// TIA Portal V15.1 export
// export: Created 2024-05-17T05:38:53.9168564Z, ExportSetting WithDefaults, DisplayName Totally Integrated Automation Portal, DisplayVersion V15.1 Update 5, DisplayName TIA Portal Openness, DisplayVersion V15.1 Update 5, DisplayName SINAMICS Startdrive Advanced, DisplayVersion V15.1, DisplayName G130, G150, S120, S150, SINAMICS MV, S210, DisplayVersion V15.1, DisplayName G110M, G120, G120C, G120D, G120P, DisplayVersion V15.1, DisplayName STEP 7 Professional, DisplayVersion V15.1 Update 5, DisplayName STEP 7 Safety, DisplayVersion V15.1, DisplayName WinCC Professional, DisplayVersion V15.1 Update 5, DisplayName SIMATIC Visualization Architect, DisplayVersion V15.1
FUNCTION_BLOCK "LVIDSRFID"   // FB1203, SCL
{ S7_Optimized_Access := 'TRUE' }
VERSION : 0.1
// stored: AutoNumber false, IsIECCheckEnabled false, IsRetainMemResEnabled false, MemoryReserve 100, SetENOAutomatically False, UDAEnableTagReadback false
   VAR_INPUT
      I_OutOfUse { ExternalAccessible := 'False'; ExternalVisible := 'False'; ExternalWritable := 'False'} : Bool;   // Module out of use
      C_AntennaTriggOnTime { ExternalAccessible := 'False'; ExternalVisible := 'False'; ExternalWritable := 'False'} : DInt := 3000;   // Default 3s
      C_AntennaTriggOffTime { ExternalAccessible := 'False'; ExternalVisible := 'False'; ExternalWritable := 'False'} : DInt := 500;   // Default 500ms
      I_AntennaStatus { ExternalAccessible := 'False'; ExternalVisible := 'False'; ExternalWritable := 'False'} : Bool;   // Antenna status
      I_StartRead { ExternalAccessible := 'False'; ExternalVisible := 'False'; ExternalWritable := 'False'} : Bool;   // On edge, start tag read
      I_InitTagEn { ExternalAccessible := 'False'; ExternalVisible := 'False'; ExternalWritable := 'False'} : Bool := FALSE;   // Init tag enabled
      I_StartInitTag { ExternalAccessible := 'False'; ExternalVisible := 'False'; ExternalWritable := 'False'} : Bool;   // On edge, start initialisation
      I_BodyIDInitTag { ExternalAccessible := 'False'; ExternalVisible := 'False'; ExternalWritable := 'False'} : DWord;   // Body identifier for init function
      I_BodyType1InitTag { ExternalAccessible := 'False'; ExternalVisible := 'False'; ExternalWritable := 'False'} : DWord;   // BodyType1
      I_PopIDInitTag { ExternalAccessible := 'False'; ExternalVisible := 'False'; ExternalWritable := 'False'} : UDInt;   // Spare Data / PopID
      I_PopIDSuffixInitTag { ExternalAccessible := 'False'; ExternalVisible := 'False'; ExternalWritable := 'False'} : Char;   // PopID suffix
      I_PopTypeInitTag { ExternalAccessible := 'False'; ExternalVisible := 'False'; ExternalWritable := 'False'} : UDInt;   // Pop identifier
      I_ResetAlarm { ExternalAccessible := 'False'; ExternalVisible := 'False'; ExternalWritable := 'False'} : Bool;   // Reset alarm
   END_VAR
   VAR_OUTPUT
      O_AntennaTrigg { ExternalAccessible := 'False'; ExternalVisible := 'False'; ExternalWritable := 'False'} : Bool;   // to antenna - start read
      O_Busy { ExternalAccessible := 'False'; ExternalVisible := 'False'; ExternalWritable := 'False'} : Bool;   // Busy
      O_ReadOK { ExternalAccessible := 'False'; ExternalVisible := 'False'; ExternalWritable := 'False'} : Bool;   // RFID read OK
      O_ReadNOK { ExternalAccessible := 'False'; ExternalVisible := 'False'; ExternalWritable := 'False'} : Bool;   // RFID read NOK
      O_InitTagBusy { ExternalAccessible := 'False'; ExternalVisible := 'False'; ExternalWritable := 'False'} : Bool;   // Tag init busy
      O_InitTagOK { ExternalAccessible := 'False'; ExternalVisible := 'False'; ExternalWritable := 'False'} : Bool;   // Tag init OK
      O_InitTagNOK { ExternalAccessible := 'False'; ExternalVisible := 'False'; ExternalWritable := 'False'} : Bool;   // Tag init NOK
      O_ReplaceTagBusy { ExternalAccessible := 'False'; ExternalVisible := 'False'; ExternalWritable := 'False'} : Bool;
      O_ReplaceTagOK { ExternalAccessible := 'False'; ExternalVisible := 'False'; ExternalWritable := 'False'} : Bool;   // Replace tag - OK
      O_ReplaceTagNOK { ExternalAccessible := 'False'; ExternalVisible := 'False'; ExternalWritable := 'False'} : Bool;   // Replace tag - NOK
      O_Status { ExternalAccessible := 'False'; ExternalVisible := 'False'; ExternalWritable := 'False'} : Int;   // Status code
      O_Alarm { ExternalAccessible := 'False'; ExternalVisible := 'False'; ExternalWritable := 'False'} : Bool;   // Alarm C / Alarm
   END_VAR
   VAR_IN_OUT
      IO_VIDS : "VIDS";   // For internal use only
      IO_VEMData : "VEMData";   // From master module
      IO_Alarm : "Alarm";   // Alarm
      H_RFID : "H_LVIDSRFID";
      H_HMI : "H_HMI";
   END_VAR
   VAR
      i { ExternalAccessible := 'False'; ExternalVisible := 'False'; ExternalWritable := 'False'} : Int;   // Index
      Reset { ExternalAccessible := 'False'; ExternalVisible := 'False'; ExternalWritable := 'False'} : Bool;
      ReadOK { ExternalAccessible := 'False'; ExternalVisible := 'False'; ExternalWritable := 'False'} : Bool;
      ReadNOK { ExternalAccessible := 'False'; ExternalVisible := 'False'; ExternalWritable := 'False'} : Bool;
      InitTagOK { ExternalAccessible := 'False'; ExternalVisible := 'False'; ExternalWritable := 'False'} : Bool;
      InitTagNOK { ExternalAccessible := 'False'; ExternalVisible := 'False'; ExternalWritable := 'False'} : Bool;
      ReplaceTagOK { ExternalAccessible := 'False'; ExternalVisible := 'False'; ExternalWritable := 'False'} : Bool;
      ReplaceTagNOK { ExternalAccessible := 'False'; ExternalVisible := 'False'; ExternalWritable := 'False'} : Bool;
      StartReplaceTagMem { ExternalAccessible := 'False'; ExternalVisible := 'False'; ExternalWritable := 'False'} : Bool;
      StartInitMem { ExternalAccessible := 'False'; ExternalVisible := 'False'; ExternalWritable := 'False'} : Bool;
      btnForceReadEdg { ExternalAccessible := 'False'; ExternalVisible := 'False'; ExternalWritable := 'False'} : Bool;
      btnForceReadPls { ExternalAccessible := 'False'; ExternalVisible := 'False'; ExternalWritable := 'False'} : Bool;
      btnInitTagByBodyIdEdg { ExternalAccessible := 'False'; ExternalVisible := 'False'; ExternalWritable := 'False'} : Bool;
      btnInitTagByBodyIdPls { ExternalAccessible := 'False'; ExternalVisible := 'False'; ExternalWritable := 'False'} : Bool;
      btnInitTagByBodyType1Edg { ExternalAccessible := 'False'; ExternalVisible := 'False'; ExternalWritable := 'False'} : Bool;
      btnInitTagByBodyType1Pls { ExternalAccessible := 'False'; ExternalVisible := 'False'; ExternalWritable := 'False'} : Bool;
      btnInitTagByPopIdEdg { ExternalAccessible := 'False'; ExternalVisible := 'False'; ExternalWritable := 'False'} : Bool;
      btnInitTagByPopIdPls { ExternalAccessible := 'False'; ExternalVisible := 'False'; ExternalWritable := 'False'} : Bool;
      btnRplcTagByMixNbrEdg { ExternalAccessible := 'False'; ExternalVisible := 'False'; ExternalWritable := 'False'} : Bool;
      btnRplcTagByMixNbrPls { ExternalAccessible := 'False'; ExternalVisible := 'False'; ExternalWritable := 'False'} : Bool;
      btnRplcTagByMixNbrEnable { ExternalAccessible := 'False'; ExternalVisible := 'False'; ExternalWritable := 'False'} : Word;
      btnRplcTagByTagIDEdg { ExternalAccessible := 'False'; ExternalVisible := 'False'; ExternalWritable := 'False'} : Bool;
      btnRplcTagByTagIDPls { ExternalAccessible := 'False'; ExternalVisible := 'False'; ExternalWritable := 'False'} : Bool;
      btnRplcTagByTagIDEnable { ExternalAccessible := 'False'; ExternalVisible := 'False'; ExternalWritable := 'False'} : Word;
      btnRplcTagByBodyIdEdg { ExternalAccessible := 'False'; ExternalVisible := 'False'; ExternalWritable := 'False'} : Bool;
      btnRplcTagByBodyIdPls { ExternalAccessible := 'False'; ExternalVisible := 'False'; ExternalWritable := 'False'} : Bool;
      btnRplcTagByBodyIdEnable { ExternalAccessible := 'False'; ExternalVisible := 'False'; ExternalWritable := 'False'} : Word;
      btnRplcTagByPopIDEdg { ExternalAccessible := 'False'; ExternalVisible := 'False'; ExternalWritable := 'False'} : Bool;
      btnRplcTagByPopIDPls { ExternalAccessible := 'False'; ExternalVisible := 'False'; ExternalWritable := 'False'} : Bool;
      btnRplcTagByPopIDEnable { ExternalAccessible := 'False'; ExternalVisible := 'False'; ExternalWritable := 'False'} : Word;
      GetVEMDataByRFIDBeginReq1 { ExternalAccessible := 'False'; ExternalVisible := 'False'; ExternalWritable := 'False'} : Bool;
      GetVEMDataByRFIDBeginReq2 { ExternalAccessible := 'False'; ExternalVisible := 'False'; ExternalWritable := 'False'} : Bool;
      GetVEMDataByRFIDBeginReq3 { ExternalAccessible := 'False'; ExternalVisible := 'False'; ExternalWritable := 'False'} : Bool;
      InteractEnable { ExternalAccessible := 'False'; ExternalVisible := 'False'; ExternalWritable := 'False'} : Bool;   // Interactions enabled
      Status { ExternalAccessible := 'False'; ExternalVisible := 'False'; ExternalWritable := 'False'} : Int;
      TriggOnTimerElapsed { ExternalAccessible := 'False'; ExternalVisible := 'False'; ExternalWritable := 'False'} : Bool;   // Antenna trigger - On
      AntennaTriggOnTimeAct { ExternalAccessible := 'False'; ExternalVisible := 'False'; ExternalWritable := 'False'} : DInt;
      TriggerOffTimerElapsed { ExternalAccessible := 'False'; ExternalVisible := 'False'; ExternalWritable := 'False'} : Bool;   // Antenna trigger - Off
      AntennaTriggOffTimeAct { ExternalAccessible := 'False'; ExternalVisible := 'False'; ExternalWritable := 'False'} : DInt;
      AntennaTrigg { ExternalAccessible := 'False'; ExternalVisible := 'False'; ExternalWritable := 'False'} : Bool;
      AntennaTriggCntr { ExternalAccessible := 'False'; ExternalVisible := 'False'; ExternalWritable := 'False'} : Int;   // Antenna trigger - Counter
      AntennaStatus { ExternalAccessible := 'False'; ExternalVisible := 'False'; ExternalWritable := 'False'} : Int;
      StartReadEdg { ExternalAccessible := 'False'; ExternalVisible := 'False'; ExternalWritable := 'False'} : Bool;
      StartReadPls { ExternalAccessible := 'False'; ExternalVisible := 'False'; ExternalWritable := 'False'} : Bool;
      StartInitTagEdg { ExternalAccessible := 'False'; ExternalVisible := 'False'; ExternalWritable := 'False'} : Bool;
      StartInitTagPls { ExternalAccessible := 'False'; ExternalVisible := 'False'; ExternalWritable := 'False'} : Bool;
      Alarm { ExternalAccessible := 'False'; ExternalVisible := 'False'; ExternalWritable := 'False'} : Bool;
      BodyIdMemReplaceTag { ExternalAccessible := 'False'; ExternalVisible := 'False'; ExternalWritable := 'False'} : DWord;
      MixNbrMemReplaceTag { ExternalAccessible := 'False'; ExternalVisible := 'False'; ExternalWritable := 'False'} : DWord;
      PopIdMemReplaceTag { ExternalAccessible := 'False'; ExternalVisible := 'False'; ExternalWritable := 'False'} : DWord;
      PopIdSuffixMemReplaceTag { ExternalAccessible := 'False'; ExternalVisible := 'False'; ExternalWritable := 'False'} : Char;
      PopTypeMemReplaceTag { ExternalAccessible := 'False'; ExternalVisible := 'False'; ExternalWritable := 'False'} : DWord;
      TagIdMem { ExternalAccessible := 'False'; ExternalVisible := 'False'; ExternalWritable := 'False'} : DWord;
      TagIdMemReplaceTag { ExternalAccessible := 'False'; ExternalVisible := 'False'; ExternalWritable := 'False'} : DWord;
      TagIdMemReplaceTagStr { ExternalAccessible := 'False'; ExternalVisible := 'False'; ExternalWritable := 'False'} : String[7];
      BodyIDMemInit { ExternalAccessible := 'False'; ExternalVisible := 'False'; ExternalWritable := 'False'} : DWord;
      BodyType1MemInit { ExternalAccessible := 'False'; ExternalVisible := 'False'; ExternalWritable := 'False'} : DWord;
      PopIDMemInit { ExternalAccessible := 'False'; ExternalVisible := 'False'; ExternalWritable := 'False'} : DWord;
      PopIDSuffixMemInit { ExternalAccessible := 'False'; ExternalVisible := 'False'; ExternalWritable := 'False'} : Char;
      PopTypeMemInit { ExternalAccessible := 'False'; ExternalVisible := 'False'; ExternalWritable := 'False'} : DWord;
      StartTriggOnTimer { ExternalAccessible := 'False'; ExternalVisible := 'False'; ExternalWritable := 'False'} : Bool;   // Trigger on timer - Start
      StartTriggOffTimer { ExternalAccessible := 'False'; ExternalVisible := 'False'; ExternalWritable := 'False'} : Bool;   // Trigger off timer - Start
      TempDiv { ExternalAccessible := 'False'; ExternalVisible := 'False'; ExternalWritable := 'False'} : DInt;   // Temporary divider
      TempDInt { ExternalAccessible := 'False'; ExternalVisible := 'False'; ExternalWritable := 'False'} : DInt;
      TempReal { ExternalAccessible := 'False'; ExternalVisible := 'False'; ExternalWritable := 'False'} : Real;
      _TriggOnTmr { ExternalAccessible := 'False'; ExternalVisible := 'False'; ExternalWritable := 'False'; S7_SetPoint := 'True'} : "LTimer";   // FB / Trigger on timer
      _TriggOffTmr { ExternalAccessible := 'False'; ExternalVisible := 'False'; ExternalWritable := 'False'; S7_SetPoint := 'True'} : "LTimer";   // FB / Trigger off timer
   END_VAR
   VAR CONSTANT
      TAG_ID_LENGTH_MAX : Int := 7;
      CMD_INIT_TAG : DWord := 2003;   // Command code - Init tag
      CMD_REPLACE_TAG : DWord := 2002;   // Command code - Replace tag
      ANTENNA_TRIGG_CNTR_MAX : Int := 3;   // Maximum amount of triggers
      STATUS_000 : Int;   // Status 000 : No action
      STATUS_001 : Int := 1;   // Status 001 : Success
      STATUS_002 : Int := 2;   // Status 002 : Busy
      STATUS_MINUS_001 : Int := -1;   // Status - 001 : No signal from RFID antenna
      STATUS_MINUS_002 : Int := -2;   // Status - 002 : Tag read error
      STATUS_MINUS_008 : Int := -12;   // Status - 008 : Sequence overtime
      STATUS_MINUS_100 : Int := -100;   // Status - 100 : TagId does not exist
      OFF : Word := 16#0000;   // HMI animation - No animation
      VISIBLE : Word := 16#0001;   // HMI animation - Visible
      ENABLE : Word := 16#0002;   // HMI animation - Enable
      COLOUR_DEFAULT : Word := 16#0000;   // HMI animation - Default colour
      COLOUR_RED : Word := 16#0010;   // HMI animation - Colour red
      COLOUR_GREEN : Word := 16#0020;   // HMI animation - Colour green
      COLOUR_BLUE : Word := 16#0040;   // HMI animation - Colour blue
      COLOUR_WHITE : Word := 16#0080;   // HMI animation - Colour white
      SECTION_HMI : Bool := TRUE;
      SECTION_OUTPUTS : Bool := TRUE;
   END_VAR
BEGIN
   (******************************************************************************
    Changelog

       17W23D1 18:00H PMo
       - Conversion from FBD TO SCL

    List OF authors

       Company : Volvo Cars Gent
       Name    : Patrick Moreau (PMo)
       E-mail  : patrick.moreau@volvocars.com
       Tel.    : +32 9 2503165

    Description

       This module is part OF the VIDS suite and is used to read, initialize and 
       replace the RFID.
       To use this module, VIDSMaster is required

    ******************************************************************************)

   (******************************************************************************)
   (* Alarm                                                                      *)
   (******************************************************************************)
   IF NOT #I_AntennaStatus AND NOT #IO_VIDS.GetVEMDataByRFID.Running AND FALSE THEN        //Check antenna
       #Status := #STATUS_MINUS_001;   //No signal from RFID antenna
   END_IF;
   IF #I_AntennaStatus AND #Status = #STATUS_MINUS_001 AND FALSE THEN
       #Status := #STATUS_000;
   END_IF;

   (******************************************************************************)
   (* Create pulses                                                              *)
   (******************************************************************************)

   //Start read - Create pulse
   #StartReadPls := #I_StartRead AND NOT #StartReadEdg;
   #StartReadEdg := #I_StartRead;

   //< Force read > button - Create pulse
   #btnForceReadPls := #H_RFID.H_btnForceRead <> 0 AND NOT #btnForceReadEdg;
   #btnForceReadEdg := #H_RFID.H_btnForceRead <> 0;

   //Start init - Create pulse
   #StartInitTagPls := #I_StartInitTag AND NOT #StartInitTagEdg;
   #StartInitTagEdg := #I_StartInitTag;

   // < Start Init tag BY BodyID > button - Create pulse
   #btnInitTagByBodyIdPls := (#H_RFID.H_btnInitTagByBodyId <> 0) AND NOT #btnInitTagByBodyIdEdg;
   #btnInitTagByBodyIdEdg := (#H_RFID.H_btnInitTagByBodyId <> 0);

   // < Start Init tag BY BodyType1 > button - Create pulse
   #btnInitTagByBodyType1Pls := (#H_RFID.H_btnInitTagByBodyType1 <> 0) AND NOT #btnInitTagByBodyType1Edg;
   #btnInitTagByBodyType1Edg := (#H_RFID.H_btnInitTagByBodyType1 <> 0);

   // < Start Init tag BY PopID > button - Create pulse
   #btnInitTagByPopIdPls := (#H_RFID.H_btnInitTagByPopId <> 0) AND NOT #btnInitTagByPopIdEdg;
   #btnInitTagByPopIdEdg := (#H_RFID.H_btnInitTagByPopId <> 0);

   //< Replace Tag BY TagID > button - Create pulse
   #btnRplcTagByTagIDPls := #H_RFID.H_btnRplcTagByTagID <> 0 AND NOT #btnRplcTagByTagIDEdg;
   #btnRplcTagByTagIDEdg := #H_RFID.H_btnRplcTagByTagID <> 0;

   //< Replace Tag BY BodyID > button - Create pulse
   #btnRplcTagByBodyIdPls := #H_RFID.H_btnRplcTagByBodyId <> 0 AND NOT #btnRplcTagByBodyIdEdg;
   #btnRplcTagByBodyIdEdg := #H_RFID.H_btnRplcTagByBodyId <> 0;

   //< Replace Tag BY Mixnumber > button - Create pulse
   #btnRplcTagByMixNbrPls := #H_RFID.H_btnRplcTagByMIxNbr <> 0 AND NOT #btnRplcTagByMixNbrEdg;
   #btnRplcTagByMixNbrEdg := #H_RFID.H_btnRplcTagByMIxNbr <> 0;

   //< Replace Tag BY PopId > button - Create pulse
   #btnRplcTagByPopIDPls := #H_RFID.H_btnRplcTagByPopId <> 0 AND NOT #btnRplcTagByPopIDEdg;
   #btnRplcTagByPopIDEdg := #H_RFID.H_btnRplcTagByPopId <> 0;

   (******************************************************************************)
   (* Get VEM data by RFID - Begin request                                       *)
   (******************************************************************************)

   //By Read
   #GetVEMDataByRFIDBeginReq1 := #I_AntennaStatus AND (#StartReadPls OR #btnForceReadPls);

   //By Replace tag
   IF  #btnRplcTagByTagIDPls THEN
       #TagIdMemReplaceTag := #H_RFID.H_txtTagIDRplcTag;
       #BodyIdMemReplaceTag := 0;
       #MixNbrMemReplaceTag := 0;
       #PopIdMemReplaceTag := 0;
       #PopIdSuffixMemReplaceTag := ' ';
       #PopTypeMemReplaceTag := 0;
       #StartReplaceTagMem := TRUE;
   ELSIF  #btnRplcTagByBodyIdPls THEN
       #TagIdMemReplaceTag := 0;
       #BodyIdMemReplaceTag := #H_RFID.H_txtBodyIDRplcTag;
       #MixNbrMemReplaceTag := 0;
       #PopIdMemReplaceTag := 0;
       #PopIdSuffixMemReplaceTag := ' ';
       #PopTypeMemReplaceTag := 0;
       #StartReplaceTagMem := TRUE;
   ELSIF  #btnRplcTagByMixNbrPls THEN
       #TagIdMemReplaceTag :=0;
       #BodyIdMemReplaceTag := 0;
       #MixNbrMemReplaceTag := #H_RFID.H_txtMixNbrRplcTag;
       #PopIdMemReplaceTag := 0;
       #PopIdSuffixMemReplaceTag := ' ';
       #PopTypeMemReplaceTag := 0;
       #StartReplaceTagMem := TRUE;
   ELSIF  #btnRplcTagByPopIDPls THEN
       #TagIdMemReplaceTag := 0;
       #BodyIdMemReplaceTag := 0;
       #MixNbrMemReplaceTag := 0;
       #PopIdMemReplaceTag := #H_RFID.H_txtPopIDRplcTag;
       #PopIdSuffixMemReplaceTag := #H_RFID.H_txtPopIDSuffixRplcTag;
       #PopTypeMemReplaceTag := #H_RFID.H_txtPopTypeRplcTag;
       #StartReplaceTagMem := TRUE;
   END_IF;
   #GetVEMDataByRFIDBeginReq2 := #btnRplcTagByTagIDPls OR #btnRplcTagByBodyIdPls OR #btnRplcTagByMixNbrPls OR #btnRplcTagByPopIDPls;

   //By Init tag
   IF  #StartInitTagPls THEN
       IF #I_BodyIDInitTag <> 0 THEN
           #BodyIDMemInit := #I_BodyIDInitTag;
           #BodyType1MemInit := 0;
           #PopIDMemInit := 0;
           #PopIDSuffixMemInit := ' ';
           #PopTypeMemInit := 0;
       ELSIF #I_BodyType1InitTag <> 0 THEN
           #BodyIDMemInit := 0;
           #PopIDMemInit := 0;
           #PopIDSuffixMemInit := ' ';
           #PopTypeMemInit := 0;
           #BodyType1MemInit := #I_BodyType1InitTag;
       ELSIF #I_PopIDInitTag <> 0 THEN
           #BodyIDMemInit := 0;
           #BodyType1MemInit := 0;
           #PopIDMemInit := #I_PopIDInitTag;
           #PopIDSuffixMemInit := #I_PopIDSuffixInitTag;
           #PopTypeMemInit := #I_PopTypeInitTag;
       END_IF;
       #StartInitMem := TRUE;
   ELSIF  #btnInitTagByBodyIdPls THEN
       #BodyIDMemInit := #H_RFID.H_txtBodyIDInitTag;
       #BodyType1MemInit := 0;
       #PopIDMemInit := 0;
       #PopIDSuffixMemInit := ' ';
       #PopTypeMemInit := 0;
       #StartInitMem := TRUE;
   ELSIF #I_AntennaStatus AND #btnInitTagByBodyType1Pls THEN
       #BodyIDMemInit := 0;
       #PopIDMemInit := 0;
       #PopIDSuffixMemInit := ' ';
       #PopTypeMemInit := 0;
       #BodyType1MemInit := #H_RFID.H_txtBodyType1InitTag;
       #StartInitMem := TRUE;
   ELSIF #I_AntennaStatus AND #btnInitTagByPopIdPls THEN
       #BodyIDMemInit := 0;
       #BodyType1MemInit := 0;
       #PopIDMemInit := #H_RFID.H_txtPopIdInitTag;
       #PopIDSuffixMemInit := #H_RFID.H_txtPopIdSuffixInitTag;
       #PopTypeMemInit := #H_RFID.H_txtPopTypeInitTag;
       #StartInitMem := TRUE;
   END_IF;

   #GetVEMDataByRFIDBeginReq3 := #StartInitTagPls OR #btnInitTagByBodyIdPls OR #btnInitTagByBodyType1Pls OR #btnInitTagByPopIdPls;

   //Begin request - Summary
   #IO_VIDS.GetVEMDataByRFID.BeginReq := #IO_VIDS.PartPres  AND
   (#GetVEMDataByRFIDBeginReq1 OR #GetVEMDataByRFIDBeginReq2 OR #GetVEMDataByRFIDBeginReq3) AND NOT 
   #IO_VIDS.GetVEMDataByRFID.Running;

   //Reset when not part present
   IF NOT #IO_VIDS.PartPres THEN

       #StartReplaceTagMem := FALSE;
       #StartInitMem := FALSE;

   END_IF;

   #Reset := NOT #IO_VIDS.PartPres OR #IO_VIDS.GetVEMDataByRFID.BeginReq OR #IO_VIDS.InitTag.BeginReq OR #IO_VIDS.ReplaceTag.BeginReq;

   IF  #Reset THEN



       #ReadOK := FALSE;
       #ReadNOK := FALSE;
       #InitTagOK := FALSE;
       #InitTagNOK := FALSE;
       #ReplaceTagOK := FALSE;
       #ReplaceTagNOK := FALSE;
       #AntennaStatus := 0;
       #Status := 0;

   END_IF;

   (******************************************************************************)
   (* Get VEM data by RFID - Begin                                               *)
   (******************************************************************************)

   //Activate antenna
   IF #IO_VIDS.GetVEMDataByRFID.OkBegin THEN
       #Status := #STATUS_002;             //Set Status busy

       #AntennaTriggCntr := 0;             //Reset antenna trigger Counter
       #StartTriggOnTimer := TRUE;         //Start trigger
   END_IF;

   //Step 0 On Active - Get VEM Data - Begin
   #IO_VIDS.GetVEMDataByRFID.Begin := #IO_VIDS.GetVEMDataByRFID.OkBegin;

   (******************************************************************************)
   (* Get VEM data by RFID - Antenna triggering                                  *)
   (******************************************************************************)

   IF NOT #I_AntennaStatus THEN
       #StartTriggOnTimer := FALSE;
       #StartTriggOffTimer := FALSE;
   END_IF;

   //Antenna Trigger on timer
   #_TriggOnTmr(I_StartTimer := #StartTriggOnTimer,
                I_HoldTimer := FALSE,
                I_MaxTimerValue := #C_AntennaTriggOnTime,
                O_TimerResult => #TriggOnTimerElapsed,
                O_TimerValue => #AntennaTriggOnTimeAct);

   //Start off timer
   IF #TriggOnTimerElapsed THEN
       #StartTriggOnTimer := FALSE;
       #StartTriggOffTimer := TRUE;
   END_IF;

   //Antenna Trigger off timer
   #_TriggOffTmr(I_StartTimer := #StartTriggOffTimer,
                 I_HoldTimer := FALSE,
                 I_MaxTimerValue := #C_AntennaTriggOffTime,
                 O_TimerResult => #TriggerOffTimerElapsed,
                 O_TimerValue => #AntennaTriggOffTimeAct);

   //Restart trigger timer
   IF #TriggerOffTimerElapsed THEN
       #AntennaTriggCntr := #AntennaTriggCntr + 1;
       IF #AntennaTriggCntr < #ANTENNA_TRIGG_CNTR_MAX THEN
           #StartTriggOffTimer := FALSE;
           #StartTriggOnTimer := TRUE;
       ELSE
           #StartTriggOnTimer := FALSE;
           #StartTriggOffTimer := FALSE;
           #AntennaStatus := #STATUS_MINUS_002;
       END_IF;
   END_IF;

   //Antenna Trigger
   #AntennaTrigg := #StartTriggOnTimer AND NOT #TriggOnTimerElapsed AND #I_AntennaStatus;

   (******************************************************************************)
   (* Get VEM data by RFID - Finish                                              *)
   (******************************************************************************)

   //Make sure we create a pulse
   #IO_VIDS.ReplaceTag.BeginReq := FALSE;
   #IO_VIDS.InitTag.BeginReq := FALSE;

   //Get VEMData by RFID - Finished
   IF #IO_VIDS.GetVEMDataByRFID.Finished THEN

       //Antenna status has priority
       IF #AntennaStatus < 0 THEN
           #Status := #AntennaStatus;
       ELSE
           #Status := #IO_VIDS.GetVEMDataByRFID.Status;
       END_IF;

       //Read OK or NOK
       IF #Status = 1 THEN
           #ReadOK := True;
       ELSE
           #ReadNOK := True;
       END_IF;

       //Replace tag
       IF #StartReplaceTagMem THEN
           #StartReplaceTagMem := FALSE;
           IF #Status <> #STATUS_MINUS_002 THEN
               #TagIdMem := #IO_VIDS.VEMData.Identification;
               #IO_VIDS.ReplaceTag.BeginReq := TRUE;       //Replace tag - Begin request
           END_IF;

       //Init tag
       ELSIF #StartInitMem THEN
           #StartInitMem := FALSE;
           IF #Status <> #STATUS_MINUS_002 THEN
               #TagIdMem := #IO_VIDS.VEMData.Identification;
               #IO_VIDS.InitTag.BeginReq := TRUE;
           END_IF;
       END_IF;

   END_IF;

   (******************************************************************************)
   (* Replace tag - Begin & Finished                                             *)
   (******************************************************************************)

   IF #IO_VIDS.ReplaceTag.OkBegin THEN

       #Status := #STATUS_002;             //Set Status busy
       #IO_VIDS.VEMData.CommandCode := #CMD_REPLACE_TAG;
       #IO_VIDS.VEMData.Identification := #TagIdMem;

       IF #TagIdMemReplaceTag <> 0 THEN
           //TagId in specificdata
           #TempDInt := DWORD_TO_DINT(#TagIdMemReplaceTag);
           #TempReal := DINT_TO_REAL(#TAG_ID_LENGTH_MAX-1);
           #TempDiv := REAL_TO_DINT(10 ** #TempReal);
           FOR #i := 0 TO (#TAG_ID_LENGTH_MAX-1) DO
               #IO_VIDS.SpecificDataInit[#i] := DINT_TO_CHAR(#TempDInt / #TempDiv + 48);
               #TempDInt := #TempDInt MOD #TempDiv;
               #TempDiv := #TempDiv / 10;
           END_FOR;
           #IO_VIDS.VEMData.SpecificDataLength := DINT_TO_DWORD(#TAG_ID_LENGTH_MAX);
       ELSE
           #IO_VIDS.VEMData.BodyID := #BodyIdMemReplaceTag;
           #IO_VIDS.VEMData.MixNumber := #MixNbrMemReplaceTag;
           #IO_VIDS.VEMData.PopID := #PopIdMemReplaceTag;
           #IO_VIDS.VEMData.PopIDSuffix := #PopIdSuffixMemReplaceTag;
           #IO_VIDS.VEMData.PopType := #PopTypeMemReplaceTag;
           #IO_VIDS.VEMData.SpecificDataLength := 0;
       END_IF;

   ELSIF #IO_VIDS.ReplaceTag.Finished THEN
       #Status := #IO_VIDS.ReplaceTag.Status;
       IF #Status = 1 THEN
           #ReplaceTagOK := True;
       ELSE
           #ReplaceTagNOK := True;
       END_IF;
   END_IF;

   #IO_VIDS.ReplaceTag.Begin := #IO_VIDS.ReplaceTag.OkBegin;

   (******************************************************************************)
   (* Init tag - Begin & Finished                                                *)
   (******************************************************************************)

   IF #IO_VIDS.InitTag.OkBegin THEN

       #Status := #STATUS_002;             //Set Status busy
       #IO_VIDS.VEMData.Identification := #TagIdMem;
       #IO_VIDS.VEMData.BodyID := #BodyIDMemInit;
       #IO_VIDS.VEMData.BodyType1 := #BodyType1MemInit;
       #IO_VIDS.VEMData.PopID := #PopIDMemInit;
       #IO_VIDS.VEMData.PopIDSuffix := #PopIDSuffixMemInit;
       #IO_VIDS.VEMData.PopType := #PopTypeMemInit;

       #IO_VIDS.VEMData.CommandCode := #CMD_INIT_TAG;

   ELSIF #IO_VIDS.InitTag.Finished THEN
       #Status := #IO_VIDS.InitTag.Status;
       IF #Status = 1 THEN
           #InitTagOK := True;
       ELSE
           #InitTagNOK := True;
       END_IF;
   END_IF;

   #IO_VIDS.InitTag.Begin := #IO_VIDS.InitTag.OkBegin;

   (******************************************************************************)
   (* Alarm = status <0                                                          *)
   (******************************************************************************)
   IF #Status < 0 THEN
       #Alarm := TRUE;
   ELSE
       #Alarm := false;
   END_IF;

   "LAlarmSummary"(I_AlarmA := "FALSE",
                   I_AlarmB := "FALSE",
                   I_AlarmC := #Alarm,
                   I_AlarmD := "FALSE",
                   I_AlarmABCondition := "FALSE",
                   IO_Alarm := #IO_Alarm,
                   C_UpperLevelHW := "FALSE",
                   C_UpperLevelSafety := "FALSE",
                   C_Safety := "FALSE",
                   C_Mechanic := "FALSE",
                   C_Transport := "FALSE",
                   C_Feature1 := "FALSE",
                   C_Feature2 := "FALSE",
                   C_Feature3 := "FALSE");

   (******************************************************************************)
   (* Outputs                                                                    *)
   (******************************************************************************)
   IF #SECTION_OUTPUTS THEN

       #O_AntennaTrigg := #AntennaTrigg;                   //Antenna Trigger

       #O_Busy := #IO_VIDS.GetVEMDataByRFID.Running;       //Read Busy
       #O_ReadOK := #ReadOK;                               //Read OK
       #O_ReadNOK := #ReadNOK;                             //Read NOK

       #O_InitTagBusy := #IO_VIDS.InitTag.Running;         //Init tag busy
       #O_InitTagOK := #InitTagOK;                         //Init OK
       #O_InitTagNOK := #InitTagNOK;                       //Init NOK

       #O_ReplaceTagBusy := #IO_VIDS.ReplaceTag.Running;   //Replace tag busy
       #O_ReplaceTagOK := #ReplaceTagOK;                   //Replace OK
       #O_ReplaceTagNOK := #ReplaceTagNOK;                 //Replace NOK

       #O_Status := #Status;                               //Status
       #O_Alarm := #Status < 0;                            //Alarm

   END_IF;
   (******************************************************************************)
   (* HMI                                                                        *)
   (******************************************************************************)

   IF #SECTION_HMI THEN

       #InteractEnable := #IO_VIDS.PartPres AND NOT #IO_VIDS.GetVEMDataByRFID.Running AND NOT #IO_VIDS.ReplaceTag.Running AND NOT #IO_VIDS.InitTag.Running;

       //HMI - IDType
       IF #IO_VIDS.IDType = 0 THEN
           #H_RFID.H_msgVEMDataBody := #VISIBLE;
           #H_RFID.H_msgVEMDataCarrier := #OFF;
       ELSE
           #H_RFID.H_msgVEMDataBody := #OFF;
           #H_RFID.H_msgVEMDataCarrier := #VISIBLE;
       END_IF;

       //HMI - Message - Part Present - Visible
       IF #IO_VIDS.PartPres THEN
           #H_RFID.H_msgPartPresAnim := #VISIBLE;
       ELSE
           #H_RFID.H_msgPartPresAnim := #OFF;
       END_IF;

       //HMI - VEM Data Valid
       IF #IO_VIDS.VEMDataValid THEN
           #H_RFID.H_msgVEMDataValidAnim := #VISIBLE;
       ELSE
           #H_RFID.H_msgVEMDataValidAnim := #OFF;
       END_IF;

       //HMI - VEM Data NOT Valid
       IF #IO_VIDS.VEMDataNotValid THEN
           #H_RFID.H_msgVEMDataNotValidAnim := #VISIBLE;
       ELSE
           #H_RFID.H_msgVEMDataNotValidAnim := #OFF;
       END_IF;

       //HMI - Status
       #H_RFID.H_msgStatus := #Status;

       //HMI - Antenna ready
       IF #I_AntennaStatus THEN
           #H_RFID.H_indReadyAnim := #VISIBLE;
       ELSE
           #H_RFID.H_indReadyAnim := #OFF;
       END_IF;

       //HMI - Read OK
       IF #ReadOK THEN
           #H_RFID.H_msgReadOkAnim := #VISIBLE;
       ELSE
           #H_RFID.H_msgReadOkAnim := 0;
       END_IF;

       //HMI - Read NOK
       IF #ReadNOK THEN
           #H_RFID.H_msgReadNokAnim := #VISIBLE;
       ELSE
           #H_RFID.H_msgReadNokAnim := 0;
       END_IF;

       //HMI - Replace tag OK
       IF #ReplaceTagOK THEN
           #H_RFID.H_msgRplcTagOkAnim := #VISIBLE;
       ELSE
           #H_RFID.H_msgRplcTagOkAnim := 0;
       END_IF;

       //HMI - Replace tag NOK
       IF #ReplaceTagNOK THEN
           #H_RFID.H_msgRplcTagNokAnim := #VISIBLE;
       ELSE
           #H_RFID.H_msgRplcTagNokAnim := 0;
       END_IF;

       //HMI - Init tag OK
       IF #InitTagOK THEN
           #H_RFID.H_msgInitTagOkAnim := #VISIBLE;
       ELSE
           #H_RFID.H_msgInitTagOkAnim := 0;
       END_IF;

       //HMI - Init tag NOK
       IF #InitTagNOK THEN
           #H_RFID.H_msgInitTagNokAnim := #VISIBLE;
       ELSE
           #H_RFID.H_msgInitTagNokAnim := 0;
       END_IF;

       //HMI - Animation Antenna Status
       IF #I_AntennaStatus THEN
           #H_RFID.H_indAntennaStatusAnim := 1;
       ELSE
           #H_RFID.H_indAntennaStatusAnim := 0;
       END_IF;

       //HMI - Animation Antenna Trigger
       IF #AntennaTrigg THEN
           #H_RFID.H_indAntennaTriggAnim := #VISIBLE;
       ELSE
           #H_RFID.H_indAntennaTriggAnim := #OFF;
       END_IF;


   (******************************************************************************)
   (* HMI - Text fields                                                          *)
   (******************************************************************************)

       //HMI - ReplaceTag - Reset Values
       IF NOT #IO_VIDS.PartPres OR (#IO_VIDS.GetVEMDataByRFID.BeginReq AND NOT #StartReplaceTagMem) THEN
           #H_RFID.H_txtTagIDRplcTag := 0;
           #H_RFID.H_txtBodyIDRplcTag := 0;
           #H_RFID.H_txtMixNbrRplcTag := 0;
           #H_RFID.H_txtPopIDRplcTag := 0;
           #H_RFID.H_txtPopIDSuffixRplcTag := ' ';
           #H_RFID.H_txtPopTypeRplcTag := 0;
       END_IF;

       IF #InteractEnable THEN
           #H_RFID.H_txtTagIDRplcTagAnim := #VISIBLE OR #ENABLE OR #COLOUR_WHITE;  //HMI - txtTagIDReplaceTag - Animation
           #H_RFID.H_txtBodyIDRplcTagAnim := #VISIBLE OR #ENABLE OR #COLOUR_WHITE;  //HMI - txtBodyIDReplaceTag - Animation
           #H_RFID.H_txtMixNbrRplcTagAnim := #VISIBLE OR #ENABLE OR #COLOUR_WHITE; //HMI - txtMixNbrReplaceTag - Animation
           #H_RFID.H_txtPopIDRplcTagAnim := #VISIBLE OR #ENABLE OR #COLOUR_WHITE; //HMI - txtPopIdReplaceTag - Animation
           #H_RFID.H_txtPopIDSuffixRplcTagAnim := #VISIBLE OR #ENABLE OR #COLOUR_WHITE; //HMI - txtPopIdSuffixReplaceTag - Animation
           #H_RFID.H_txtPopTypeRplcTagAnim := #VISIBLE OR #ENABLE OR #COLOUR_WHITE; //HMI - txtPopTypeReplaceTag - Animation
       ELSE
           #H_RFID.H_txtTagIDRplcTagAnim := #VISIBLE OR #COLOUR_DEFAULT;  //HMI - txtTagIDReplaceTag - Animation
           #H_RFID.H_txtBodyIDRplcTagAnim := #VISIBLE OR #COLOUR_DEFAULT;  //HMI - txtBodyIDReplaceTag - Animation
           #H_RFID.H_txtMixNbrRplcTagAnim := #VISIBLE OR #COLOUR_DEFAULT; //HMI - txtMixNbrReplaceTag - Animation
           #H_RFID.H_txtPopIDRplcTagAnim := #VISIBLE OR #COLOUR_DEFAULT; //HMI - txtPopIdReplaceTag - Animation
           #H_RFID.H_txtPopIDSuffixRplcTagAnim := #VISIBLE OR #COLOUR_DEFAULT; //HMI - txtPopIdSuffixReplaceTag - Animation
           #H_RFID.H_txtPopTypeRplcTagAnim := #VISIBLE OR #COLOUR_DEFAULT; //HMI - txtPopTypeReplaceTag - Animation
       END_IF;


       //HMI - InitTag - Reset Values
       IF NOT #IO_VIDS.PartPres OR (#IO_VIDS.GetVEMDataByRFID.BeginReq AND NOT #StartInitMem) THEN
           #H_RFID.H_txtBodyIDInitTag := 0;
           #H_RFID.H_txtBodyType1InitTag := 0;
           #H_RFID.H_txtPopIdInitTag := 0;
           #H_RFID.H_txtPopIdSuffixInitTag := ' ';
           #H_RFID.H_txtPopTypeInitTag := 0;
       END_IF;

       //HMI - InitTag
       IF #I_InitTagEn  THEN
           IF #InteractEnable THEN
               #H_RFID.H_txtBodyIDInitTagAnim := #VISIBLE OR #ENABLE OR #COLOUR_WHITE;     //HMI - txtBodyIDInitTag - Animation
               #H_RFID.H_txtBodyType1InitTagAnim := #VISIBLE OR #ENABLE OR #COLOUR_WHITE;  //HMI - txtBodyType1InitTag - Animation
               #H_RFID.H_txtPopIdInitTagAnim := #VISIBLE OR #ENABLE OR #COLOUR_WHITE;      //HMI - txtPopIdInitTag - Animation
               #H_RFID.H_txtPopIdSuffixInitTagAnim := #VISIBLE OR #ENABLE OR #COLOUR_WHITE;//HMI - txtPopIdSuffixInitTag - Animation
               #H_RFID.H_txtPopTypeInitTagAnim := #VISIBLE OR #ENABLE OR #COLOUR_WHITE;    //HMI - txtPopTypeInitTag - Animation
           ELSE
               #H_RFID.H_txtBodyIDInitTagAnim := #VISIBLE OR #COLOUR_DEFAULT;     //HMI - txtBodyIDInitTag - Animation
               #H_RFID.H_txtBodyType1InitTagAnim := #VISIBLE OR #COLOUR_DEFAULT;  //HMI - txtBodyType1InitTag - Animation
               #H_RFID.H_txtPopIdInitTagAnim := #VISIBLE OR #COLOUR_DEFAULT;      //HMI - txtPopIdInitTag - Animation
               #H_RFID.H_txtPopIdSuffixInitTagAnim := #VISIBLE OR #COLOUR_DEFAULT;//HMI - txtPopIdSuffixInitTag - Animation
               #H_RFID.H_txtPopTypeInitTagAnim := #VISIBLE OR #COLOUR_DEFAULT;    //HMI - txtPopTypeInitTag - Animation
           END_IF;
       ELSE
           #H_RFID.H_txtBodyIDInitTagAnim := #VISIBLE;         //HMI - txtBodyIDInitTag - Animation
           #H_RFID.H_txtBodyType1InitTagAnim := #VISIBLE;      //HMI - txtBodyType1InitTag - Animation
           #H_RFID.H_txtPopIdInitTagAnim := #VISIBLE;          //HMI - txtPopIdInitTag - Animation
           #H_RFID.H_txtPopIdSuffixInitTagAnim := #VISIBLE;    //HMI - txtPopIdSuffixInitTag - Animation
           #H_RFID.H_txtPopTypeInitTagAnim := #VISIBLE;        //HMI - txtPopTypeInitTag - Animation
       END_IF;

       //VEM data

       #H_RFID.H_txtTagID := #IO_VEMData.Identification;
       #H_RFID.H_txtBodyID := #IO_VEMData.BodyID;                          //HMI - txtBodyNbr - Value
       #H_RFID.H_txtMixNbr := #IO_VEMData.MixNumber;                       //HMI - txtMixnNbr - Value
       #H_RFID.H_txtCarrierID := #IO_VEMData.CarrierID;                    //HMI - txtCarrierID - Value
       #H_RFID.H_txtBodyTypeMatrix := #IO_VEMData.BodyTypeMatrix;          //HMI - txtBodyTypeMatrix - Value
       #H_RFID.H_txtBodyType1 := #IO_VEMData.BodyType1;                    //HMI - txtBodyType1 - Value
       #H_RFID.H_txtPopId := #IO_VEMData.PopID;                            //HMI - txtPopID - Value
       #H_RFID.H_txtPopIdSuffix := #IO_VEMData.PopIDSuffix;                //HMI - txtPopID - Value
       #H_RFID.H_txtPopType := #IO_VEMData.PopType;                        //HMI - txtPopType - Value

       #H_RFID.H_txtCommandCodeSent := #IO_VIDS.CmdCodeSent;               //HMI - CmdCode Sent
       #H_RFID.H_txtCommandCodeRcvd := #IO_VIDS.CmdCodeRcvd;               //HMI - CmdCode Received

   (******************************************************************************)
   (* HMI - Buttons                                                              *)
   (******************************************************************************)

       #H_RFID.H_btnForceReadAnim := #VISIBLE OR #ENABLE;

       //Replace tag
       IF #H_RFID.H_txtTagIDRplcTag <> 0 THEN
           #btnRplcTagByTagIDEnable := #ENABLE;
       ELSE
           #btnRplcTagByTagIDEnable := #OFF;
       END_IF;
       #H_RFID.H_btnRplcTagByTagIDAnim := #VISIBLE OR #btnRplcTagByTagIDEnable;

       //Replace tag
       IF #H_RFID.H_txtBodyIDRplcTag <> 0 THEN
           #btnRplcTagByBodyIdEnable := #ENABLE;
       ELSE
           #btnRplcTagByBodyIdEnable := #OFF;
       END_IF;
       #H_RFID.H_btnRplcTagByBodyIdAnim := #VISIBLE OR #btnRplcTagByBodyIdEnable;

       //Replace tag
       IF #H_RFID.H_txtMixNbrRplcTag <> 0 THEN
           #btnRplcTagByMixNbrEnable := #ENABLE;
       ELSE
           #btnRplcTagByMixNbrEnable := #OFF;
       END_IF;
       #H_RFID.H_btnRplcTagByMixNbrAnim := #VISIBLE OR #btnRplcTagByMixNbrEnable;

       //Replace tag
       IF #H_RFID.H_txtPopIDRplcTag <> 0 THEN
           #btnRplcTagByPopIDEnable := #ENABLE;
       ELSE
           #btnRplcTagByPopIDEnable := #OFF;
       END_IF;
       #H_RFID.H_btnRplcTagByPopIdAnim := #VISIBLE OR #btnRplcTagByPopIDEnable;

       //Init tag
       IF #I_InitTagEn THEN
           #H_RFID.H_btnInitTagByBodyIdAnim := #VISIBLE OR #ENABLE;
           #H_RFID.H_btnInitTagByBodyType1Anim := #VISIBLE OR #ENABLE;
           #H_RFID.H_btnInitTagByPopIdAnim := #VISIBLE OR #ENABLE;
       ELSE
           #H_RFID.H_btnInitTagByBodyIdAnim := #VISIBLE;
           #H_RFID.H_btnInitTagByBodyType1Anim := #VISIBLE;
           #H_RFID.H_btnInitTagByPopIdAnim := #VISIBLE;
       END_IF;

       //HMI Reset buttons
       #H_RFID.H_btnForceRead := 0;
       #H_RFID.H_btnRplcTagByTagID := 0;
       #H_RFID.H_btnRplcTagByBodyId := 0;
       #H_RFID.H_btnRplcTagByMIxNbr := 0;
       #H_RFID.H_btnRplcTagByPopId := 0;
       #H_RFID.H_btnInitTagByBodyId := 0;
       #H_RFID.H_btnInitTagByBodyType1 := 0;
       #H_RFID.H_btnInitTagByPopId := 0;

   (******************************************************************************)
   (* Icon animation                                                             *)
   (******************************************************************************)

       "LIAnimDWord"(I_SetPos := FALSE,
                     I_ResetPos := FALSE,
                     I_Active := #Status > 1,
                     I_Visible := FALSE,
                     I_OutOfUse := FALSE,
                     I_IntlkSet := FALSE,
                     I_IntlkReset := FALSE,
                     I_IntlkSetAlm := FALSE,
                     I_IntlkResetAlm := FALSE,
                     I_ManualMode := FALSE,
                     I_FncSelInHMI := FALSE,
                     I_AnySelected := FALSE,
                     I_AlarmA := FALSE,
                     I_AlarmB := FALSE,
                     I_AlarmC := #Status < 0,
                     I_AlarmD := FALSE,
                     I_SafetyOk := FALSE,
                     I_Service:="TRUE",
                     I_Spare1:="FALSE",
                     I_Spare2:="FALSE",
                     I_Spare3:="FALSE",
                     I_Spare4:="FALSE",
                     I_Spare5:="FALSE",
                     I_Spare6:="FALSE",
                     I_Spare7:="FALSE",
                     I_Spare8:="FALSE",
                     I_Spare9:="FALSE",
                     I_Spare10:="FALSE",
                     I_Spare11:="FALSE",
                     I_Spare12:="FALSE",
                     I_Spare13:="FALSE",
                     I_Spare14:="FALSE",
                     H_IAnim => #H_HMI.H_IAnim);

   END_IF;
END_FUNCTION_BLOCK
